// TIA Portal V18 export
DATA_BLOCK "CAB_yLEDALARM_DB"   // DB45
VERSION : 0.1
// stored: AutoNumber true, DBAccessibleFromOPCUA true, InstanceOfName LED_FBD, InstanceOfType FB
"LED_FBD"
   // VAR_INPUT
   //    on : Bool;
   //    blink : Bool;
   //    t_on : Time;
   //    t_off : Time;
   //    ignoreTestAll : Bool;
   // END_VAR
   // VAR_OUTPUT
   //    y : Bool;
   // END_VAR
   // VAR_IN_OUT
   //    testHMI : Bool;
   // END_VAR
   // VAR
   //    blink1 { S7_SetPoint := 'True'} : "BLINKER";
   //    blink_st : Bool;
   //    tonhmi { S7_SetPoint := 'True'} : TON_TIME;
   // END_VAR
BEGIN
END_DATA_BLOCK
